FUNCTION_BLOCK FB_CNV
VAR_INPUT
	// Steuereingänge
	bEnable : BOOL;
	bExecute : BOOL;
	bHalt : BOOL;
	//Bewegungseigenschaften
	rVel : REAL;
END_VAR
VAR_OUTPUT
	eState : E_State;
END_VAR
VAR
	nState : INT;
	mcPower : MC_Power;
	mcReset : MC_Reset;
	mcVelocity : MC_MoveVelocity;
	mcHalt : MC_Halt;
	mcStop : MC_Stop;
	bStop : BOOL;
END_VAR
VAR_IN_OUT
	ax : Axis_Ref;
END_VAR

// Fehlerüberwachung
IF ax.Status.Error AND nState <> 100 THEN
    nState := 99;
END_IF

bStop := ifc_Hw.bStop;

// States
CASE nState OF
    0: // Off
        eState := E_State.Off;
        mcPower.Enable := FALSE;
        mcPower.Enable_Positive := FALSE;
        mcPower.Enable_Negative := FALSE;
        mcVelocity.Execute := FALSE;
        mcHalt.Execute := FALSE;
        mcReset.Execute := FALSE;
        
        IF bEnable THEN
            nState := 1;
        END_IF
		
		
        
    1: // Init 
        eState := E_State.Init;
        mcPower.Enable := TRUE;
        mcPower.Enable_Positive := TRUE;
        mcPower.Enable_Negative := TRUE;
        
        IF mcPower.Status THEN // State übergang
            nState := 2;
        END_IF
        
        // abbruch
        IF NOT bEnable THEN nState := 0; END_IF 
        
    2: // Ready 
        eState := E_State.Ready;
        mcVelocity.Execute := FALSE;
        mcHalt.Execute := FALSE;
        
        IF bExecute THEN
            nState := 3; // State übergang
        END_IF
        
        // abbruch
        IF NOT bEnable THEN nState := 0; END_IF 
        
    3: // CNV an 
        eState := E_State.Production;
        mcVelocity.Velocity := rVel;
        mcVelocity.Direction := MC_Positive_Direction;
        mcVelocity.Execute := TRUE;
        
        // abbruch mit abbremsen
        IF bHalt OR NOT bEnable THEN
            nState := 4;
        END_IF
        
    4: // CNV aus 
        eState := E_State.Production;
        mcVelocity.Execute := FALSE;
        mcHalt.Execute := TRUE; // Bremsvorgang einleiten
        
        IF mcHalt.Done THEN 
            nState := 5;
        END_IF
        
    5: // Done 
        eState := E_State.Done;
        mcHalt.Execute := FALSE;
        
        IF NOT bEnable THEN
            nState := 0; 
        ELSIF NOT bExecute AND NOT bHalt THEN
            nState := 2; // Wieder zurück auf Ready
        END_IF
		
	80: // Stop CNV
		mcVelocity.Execute := FALSE;
		mcHalt.Execute := FALSE;
		mcStop.Execute := TRUE;
		
		IF mcStop.Done AND NOT bStop THEN
			nState := 81;
		END_IF
        
	81: 
		mcVelocity.Execute := FALSE;
		mcHalt.Execute := FALSE;
		mcStop.Execute := TRUE;
		mcReset.Execute := TRUE;
		
		IF mcReset.Done THEN
			nState := 3;
		END_IF
	
    99: // Error State
        eState := E_State.Error;
        mcPower.Enable := FALSE;
        mcPower.Enable_Positive := FALSE;
        mcPower.Enable_Negative := FALSE;
        mcVelocity.Execute := FALSE;
        mcHalt.Execute := FALSE;
        
        IF bEnable THEN 
            nState := 100;
        END_IF
        
    100: // Resolve 
        mcReset.Execute := TRUE;
        
        IF mcReset.Done THEN
            mcReset.Execute := FALSE;
            nState := 1; // Neustart nach Reset
        ELSIF mcReset.Error THEN
            mcReset.Execute := FALSE;
            nState := 99; // Reset fehlgeschlagen
        END_IF
        
END_CASE

// Bausteine aufrufen
mcPower(Axis := ax, Enable := mcPower.Enable, Enable_Positive := mcPower.Enable_Positive, Enable_Negative := mcPower.Enable_Negative, Override := 100.0);
mcReset(Axis := ax, Execute := mcReset.Execute);
mcVelocity(Axis := ax, Execute := mcVelocity.Execute, Velocity := mcVelocity.Velocity, Direction := mcVelocity.Direction);
mcHalt(Axis := ax, Execute := mcHalt.Execute);

END_FUNCTION_BLOCK

(* stored: Version 1.1.0.1
   POU FB_CNV: Id {bede6ce1-2426-4b38-8842-9ecb657cee19}, SpecialFunc None *)
